// TIA Portal V20 export
TYPE "type_emRelations_em6_sequence"
// stored: Access Published, Namespace Unit1
   STRUCT
      hotPressLeft : Struct
         jobs : "LAF_typeJobs";
         sequence : "LAF_typeSequence";
         selectJobStatus { S7_SetPoint := 'True'} : Array[0..10] of "LAF_typeJobStatus";
         "step" : "LER_typeStep";
         jobInterface : Struct
            loadJob2 : "LER_typeJobInterface";
            inspectionJob3 : "LER_typeJobInterface";
            unloadJob4 : "LER_typeJobInterface";
         END_STRUCT;
         homeCheck : Struct
            liftDownPartNoDetect : Bool;
            liftDownPartDetect : Bool;
            liftUp : Bool;
         END_STRUCT;
      END_STRUCT;
   END_STRUCT;
   // // hotPressLeft."step".action1[101] : Step[101] : JOB[1] Condition
   // // hotPressLeft."step".action1[110] : Step[110] : Servo Press Reference Home Pos
   // // hotPressLeft."step".action1[120] : Step[120] : Spare
   // // hotPressLeft."step".action1[130] : Step[130] : Spare
   // // hotPressLeft."step".action1[140] : Step[140] : Spare
   // // hotPressLeft."step".action1[160] : Step[160] : Stage Lift Down
   // // hotPressLeft."step".action1[170] : Step[170] : Spare
   // // hotPressLeft."step".action1[190] : Step[190] : JOB[1] Step End
   // // hotPressLeft."step".action1[201] : Step[201] : JOB[2] Condition
   // // hotPressLeft."step".action1[210] : Step[210] : Hot Press Left Loading Request => Transfer PP Left
   // // hotPressLeft."step".action1[220] : Step[220] : Spare
   // // hotPressLeft."step".action1[230] : Step[230] : Stage Lift Up
   // // hotPressLeft."step".action1[240] : Step[240] : Hot Press Left Loading Check => Transfer PP Left
   // // hotPressLeft."step".action1[250] : Step[250] : Spare
   // // hotPressLeft."step".action1[290] : Step[290] : JOB[2] Step End
   // // hotPressLeft."step".action1[301] : Step[301] : JOB[3] Condition
   // // hotPressLeft."step".action1[310] : Step[310] : Stage Lift Down
   // // hotPressLeft."step".action1[311] : Step[311] : Stage JR Detection Check
   // // hotPressLeft."step".action1[320] : Step[320] : Spare
   // // hotPressLeft."step".action1[330] : Step[330] : Hot Press Start
   // // hotPressLeft."step".action1[331] : Step[331] : Hot Press Result
   // // hotPressLeft."step".action1[380] : Step[380] : Hot Press Home Return
   // // hotPressLeft."step".action1[390] : Step[390] : JOB[3] Step End
   // // hotPressLeft."step".action1[401] : Step[401] : JOB[4] Condition
   // // hotPressLeft."step".action1[410] : Step[410] : Spare
   // // hotPressLeft."step".action1[420] : Step[420] : Stage Lift Up
   // // hotPressLeft."step".action1[430] : Step[430] : Hot Press Left Unloading Request => Transfer PP Left
   // // hotPressLeft."step".action1[431] : Step[431] : Hot Press Left Unloading Check => Transfer PP Left
   // // hotPressLeft."step".action1[480] : Step[480] : Stage Lift Down
   // // hotPressLeft."step".action1[481] : Step[481] : Spare
   // // hotPressLeft."step".action1[490] : Step[490] : JOB[4] Step End
   // // hotPressLeft."step".transition1[101] : Step[101] : JOB[1] Condition
   // // hotPressLeft."step".transition1[110] : Step[110] : Servo Press Reference Home Pos
   // // hotPressLeft."step".transition1[120] : Step[120] : Spare
   // // hotPressLeft."step".transition1[130] : Step[130] : Spare
   // // hotPressLeft."step".transition1[140] : Step[140] : Spare
   // // hotPressLeft."step".transition1[160] : Step[160] : Stage Lift Down
   // // hotPressLeft."step".transition1[170] : Step[170] : Spare
   // // hotPressLeft."step".transition1[190] : Step[190] : JOB[1] Step End
   // // hotPressLeft."step".transition1[201] : Step[201] : JOB[2] Condition
   // // hotPressLeft."step".transition1[210] : Step[210] : Hot Press Left Loading Request => Transfer PP Left
   // // hotPressLeft."step".transition1[220] : Step[220] : Spare
   // // hotPressLeft."step".transition1[230] : Step[230] : Stage Lift Up
   // // hotPressLeft."step".transition1[240] : Step[240] : Hot Press Left Loading Check => Transfer PP Left
   // // hotPressLeft."step".transition1[250] : Step[250] : Spare
   // // hotPressLeft."step".transition1[290] : Step[290] : JOB[2] Step End
   // // hotPressLeft."step".transition1[301] : Step[301] : JOB[3] Condition
   // // hotPressLeft."step".transition1[310] : Step[310] : Stage Lift Down
   // // hotPressLeft."step".transition1[311] : Step[311] : Stage JR Detection Check
   // // hotPressLeft."step".transition1[320] : Step[320] : Spare
   // // hotPressLeft."step".transition1[330] : Step[330] : Hot Press Start
   // // hotPressLeft."step".transition1[331] : Step[331] : Hot Press Result
   // // hotPressLeft."step".transition1[380] : Step[380] : Hot Press Home Return
   // // hotPressLeft."step".transition1[390] : Step[390] : JOB[3] Step End
   // // hotPressLeft."step".transition1[401] : Step[401] : JOB[4] Condition
   // // hotPressLeft."step".transition1[410] : Step[410] : Spare
   // // hotPressLeft."step".transition1[420] : Step[420] : Stage Lift Up
   // // hotPressLeft."step".transition1[430] : Step[430] : Hot Press Left Unloading Request => Transfer PP Left
   // // hotPressLeft."step".transition1[431] : Step[431] : Hot Press Left Unloading Check => Transfer PP Left
   // // hotPressLeft."step".transition1[480] : Step[480] : Stage Lift Down
   // // hotPressLeft."step".transition1[481] : Step[481] : Spare
   // // hotPressLeft."step".transition1[490] : Step[490] : JOB[4] Step End
END_TYPE
